TYPE stParam_Counter :
STRUCT
	WrittenFor: STRING := '';
	nMax: UINT := 6;
END_STRUCT
END_TYPE

(* stored: Version 1.1.0.1, ProductVersion 3.1.4026.18
   DUT stParam_Counter: Id {67e2d41b-8a60-42bb-8846-3396c4b3b181} *)
